{attribute 'pack_mode' := '1'} 
TYPE ST_TxRxMessage :
STRUCT
	dataLength : UINT;
	cobId : UDINT;
	data : ARRAY[0..7] OF BYTE;
END_STRUCT
END_TYPE

(* stored: Version 1.1.0.1, ProductVersion 3.1.4024.11
   DUT ST_TxRxMessage: Id {70a31e72-34b7-44d5-ba7e-f68c2480e118} *)
